FUNCTION_BLOCK POU1
VAR_INPUT
END_VAR
VAR_OUTPUT
END_VAR
VAR
END_VAR

END_FUNCTION_BLOCK

(* stored: Version 1.1.0.1, ProductVersion 3.1.4020.12
   POU POU1: Id {b61f3b3c-423f-4aac-b3bd-74075572c7bb}, SpecialFunc None *)
